// TIA Portal V19 export
VAR_GLOBAL   // PLC tag table "Default tag table"
   memSensorType2 AT %MW14 : Int;
   memSensorType1 AT %MW16 : Int;
   Tag_1 AT %T5 : Timer;
END_VAR
VAR_GLOBAL CONSTANT   // user constants
   PANELS_NO : Int := 2;
   LACYCCOM_BUFFER_ELEMENTS_UPPER_LIM : Int := 59;   // Upper limit of request buffer array
   LACYCCOM_WRITE_PARAMETERS_UPPER_LIM : Int := 18;   // Upper limit of write parameters
   LACYCCOM_READ_PARAMETERS_UPPER_LIM : Int := 38;   // Upper limit of read parameters
   LACYCCOM_SILENT_OPERATION_PARAMETERS_UPPER_LIM : Int := 17;   // Upper limit of parameters in LAcycCom_typeDriveSilentOperation
   LACYCCOM_NO_COMMAND : Byte := 16#00;   // No command
   LACYCCOM_READ_COMMAND : Byte := 16#01;   // Read command
   LACYCCOM_WRITE_COMMAND : Byte := 16#02;   // Write command
   LACYCCOM_TYPE_ALARM : SInt := 1;   // Alarm
   LACYCCOM_TYPE_FAULT : SInt := 2;   // Fault
   LACYCCOM_TYPE_SI_MESSAGE : SInt := 3;   // SI message
   LACYCCOM_MESSAGES_UPPER_LIM : Int := 23;   // Upper limit of elements in LAcycCom_typeDriveMessages (fix value)
END_VAR
